// Mitsubishi GX Works2 project: project   PLC: FX3U/FX3UC
// Okoma

TYPE spindleProfile : STRUCT
  valveUp : BOOL;  (* DO_ Valve to move spindle UP *)
  valveDown : BOOL;  (* DO_ Valve to move spindle DOWN *)
  valveInMan : BOOL;  (* Command from HMI to move spindle IN/OUT work *)
  motorOnMan : BOOL;  (* Command from HMI to switch ON motor *)
  recipeOn : BOOL;  (* Spindle must be ON by Recipe from HMI *)
  recipeUp : BOOL;  (* Spindle must be UP by Recipe from HMI *)
  valveUpMan : BOOL;  (* Command from HMI to move spindle UP *)
  valveDownMan : BOOL;  (* Command from HMI to move spindle DOWN *)
  valveIn : BOOL;  (* DO_ Valve to move spindle IN work *)
  motorOn : BOOL;  (* DO_ Contactor to switch ON motor *)
  sensorUp : BOOL;  (* DI_ Sensor spindle in Top position *)
  sensorDown : BOOL;  (* DI_ Sensor spindle in Bottom position *)
  sensorOut : BOOL;  (* DI_ Sensor spindle position OUT of work *)
END_STRUCT END_TYPE

// global labels: Global_Vars
VAR_GLOBAL
  hmiPar10 AT D200.0 : BOOL;  (* Return after Quick Cut Cycle (0-Off, 1-On) *)
  recipeRollerPresser AT D250.4 : BOOL;
  recipeMotor0 AT D250.5 : BOOL;
  recipeMotor4 AT D250.9 : BOOL;
  recipeMotor5 AT D250.A : BOOL;
  recipeBlower AT D250.B : BOOL;
  recipeBetween2and3 AT D250.F : BOOL;
  recipeSpindle0bit0 AT D251.0 : BOOL;
  recipeSpindle0bit1 AT D251.1 : BOOL;
  safetyCircuiteOk AT M0 : BOOL;
  automaticMode AT M5 : BOOL;
  manualMode AT M6 : BOOL;
  alarmState AT M7 : BOOL;
  attentionState AT M8 : BOOL;
  spindle0NotMiddle AT M10 : BOOL;
  carriageBlockNotChange AT M12 : BOOL;
  spindle0NotChange AT M11 : BOOL;
  motorsProfile AT M40 : BOOL;  (* Motor 1, 2,3 or 5 (saw end) is ON *)
  rollersTransporterAuto AT M30 : BOOL;
  carriageMoving AT M20 : BOOL;
  machineBusy AT M9 : BOOL;  (* Excecutung automatic cycle *)
  manCarriageMoveToSensor4 AT M24 : BOOL;
  manCarriageMoveToSensor1 AT M25 : BOOL;
  rollersTransporterContinousMan AT M31 : BOOL;
  thermicOk AT X000 : BOOL;
  controlVoltageOk AT X001 : BOOL;
  airPressureOk AT X002 : BOOL;
  bypassKey AT X003 : BOOL;
  buttonQuickCut AT X010 : BOOL;
  buttonPositioningSpindles AT X017 : BOOL;  (* button S3 *)
  buttonStart2 AT X020 : BOOL;
  carriageSensor1 AT X021 : BOOL;
  carriageSensor2 AT X022 : BOOL;
  carriageSensor3 AT X023 : BOOL;
  carriageSensor4 AT X024 : BOOL;
  pieceInStart AT X025 : BOOL;
  pieceInEnd AT X026 : BOOL;
  buttonStartMotors AT X027 : BOOL;  (* button S60 *)
  buttonAuto AT X030 : BOOL;  (* button S55 *)
  buttonPress AT X031 : BOOL;  (* button S54 *)
  buttonStart AT X032 : BOOL;  (* button S53 *)
  buttonEnable AT X033 : BOOL;  (* button S61 *)
  buttonTransporterForward AT X034 : BOOL;  (* button S62 *)
  buttonTransporterBackward AT X035 : BOOL;  (* button S63 *)
  buttonCarriageForward AT X036 : BOOL;  (* button S36 *)
  buttonCarriageBackward AT X037 : BOOL;  (* button S37 *)
  carriageMoveEnable AT Y001 : BOOL;
  carriageMotorForward AT Y002 : BOOL;
  carriageMotorBackward AT Y003 : BOOL;
  carriageMotorBrake AT Y004 : BOOL;  (* Brake resistor *)
  carriageSpeedWork AT Y005 : BOOL;
  carriageSpeedSlow AT Y006 : BOOL;
  carriageSpeedFast AT Y007 : BOOL;
  spindleMotor0 AT Y010 : BOOL;  (* Motor 0 *)
  sawCarriageMotor AT Y014 : BOOL;  (* Motor 4 *)
  sawEndMotor AT Y015 : BOOL;  (* Motor 5 *)
  transporterMotorBackward AT Y016 : BOOL;
  transporterMotorForward AT Y017 : BOOL;
  pressCarriageValveDown AT Y020 : BOOL;
  spindle0Valve1Up AT Y024 : BOOL;
  spindle0Valve1Down AT Y025 : BOOL;
  spindle0Valve2Up AT Y026 : BOOL;
  spindle0Valve2Down AT Y027 : BOOL;
  pressCarriageValveUp AT Y030 : BOOL;
  pressRollerReleaseValve AT Y037 : BOOL;
  between2and3Valve AT Y040 : BOOL;
  blower AT Y041 : BOOL;
  sawEndValveDown AT Y042 : BOOL;
  lightAlarm AT Y044 : BOOL;
  lightCycleRun AT Y045 : BOOL;  (* Automatic Cycle running White indicator *)
  lightAttention AT Y046 : BOOL;
  PLC_Run AT M8000 : BOOL;
  PLC_getErrors AT M8004 : BOOL;
  carriageNeedForward AT M27 : BOOL;
  carriageNeedBackward AT M28 : BOOL;
  Alarm52 AT D5.2 : BOOL;  (* Alarm: Start Automtic cycle with all motors off *)
  Alarm53 AT D5.3 : BOOL;  (* Alarm: Piece not fixed on carriage by press *)
  Alarm54 AT D5.4 : BOOL;  (* Alarm: Change state motors while some cycle is running *)
  Alarm55 AT D5.5 : BOOL;  (* Alarm: Start motors not in Automatic mode *)
  Alarm46 AT D4.6 : BOOL;  (* Alarm: Too long time Carriage moving backward *)
  Alarm01 AT D0.1 : BOOL;  (* Alarm: Thermic breakers KO *)
  Alarm02 AT D0.2 : BOOL;  (* Alarm: Low air pressure *)
  Alarm03 AT D0.3 : BOOL;  (* Alarm: Control voltage KO *)
  Alarm04 AT D0.4 : BOOL;  (* Alarm: Stop button pressed *)
  Alarm09 AT D0.9 : BOOL;  (* Alarm: Bypass key switched on *)
  Alarm11 AT D1.1 : BOOL;  (* Alarm: Spindle 1 Top and buttom sensors ON *)
  Alarm12 AT D1.2 : BOOL;  (* Alarm: Spindle 1 not in horisontal position *)
  Alarm13 AT D1.3 : BOOL;  (* Alarm: Spindle 1 not in vertical position *)
  Alarm21 AT D2.1 : BOOL;  (* Alarm: Spindle 2 Top and Buttom sensors ON *)
  Alarm22 AT D2.2 : BOOL;  (* Alarm: Spindle 2 not in horisontal position *)
  Alarm23 AT D2.3 : BOOL;  (* Alarm: Spindle 2 not in vertical position *)
  Alarm31 AT D3.1 : BOOL;  (* Alarm: Spindle 3 Top and buttom sensors ON *)
  Alarm32 AT D3.2 : BOOL;  (* Alarm: Spindle 3 Not in horisontal position *)
  Alarm33 AT D3.3 : BOOL;  (* Alarm: Spindle 3 Not in vertical position *)
  Alarm40 AT D4.0 : BOOL;  (* Alarm: More than one carriage sensor ON in one time *)
  Alarm45 AT D4.5 : BOOL;  (* Alarm: Too long time Carriage moving forward *)
  Alarm56 AT D5.6 : BOOL;  (* Alarm: Positioning spindles not in Automatic mode *)
  Alarm47 AT D4.7 : BOOL;  (* Alarm: Move carriage with Spindle 0 in middle *)
  Alarm58 AT D5.8 : BOOL;  (* Alarm: Positioning spindles 0 with block change and piece pressed *)
  Alarm59 AT D5.9 : BOOL;  (* Alarm: Positioning spindles 0 in carriage unknown position *)
  Alarm50 AT D5.0 : BOOL;  (* Alarm: Positionig cycle by pneumatic not finished *)
  Alarm51 AT D5.1 : BOOL;  (* Alarm: Start motors cycle not finished *)
  motorsDovetail AT M41 : BOOL;  (* Motor 0 or 4 (saw carriage) is ON *)
  Alarm57 AT D5.7 : BOOL;  (* Alarm: Positioning spindles while some cycle is running *)
  Alarm5A AT D5.A : BOOL;  (* Alarm: Start cycle not in Automatic mode *)
  Alarm5C AT D5.C : BOOL;  (* Alarm: Start Automatic cycle while another cycle is running *)
  PLC_InitialPulse AT M8002 : BOOL;
  Alarm48 AT D4.8 : BOOL;  (* Alarm: Move carriage backward with Sensor 1 On *)
  Alarm49 AT D4.9 : BOOL;  (* Alarm: Move carriage forward with Sensor 4 On *)
  plcRunTime AT D10 : TIME;  (* PLC running time in ms (step 10 ms) *)
  hmiPar11 AT D200.1 : BOOL;  (* Cut (0-slow, 1-quick) *)
  workTime AT D230 : DINT;  (* Time machine run (in seconds) *)
  hmiPar1 AT D201 : TIME;  (* Delay to slowdown carriage (0..5sec) *)
  hmiPar2 AT D203 : TIME;
  hmiPar3 AT D205 : TIME;  (* Delay carriage presser release (0..1sec) *)
  hmiPar4 AT D207 : TIME;  (* Delay blower OFF (0..60sec) *)
  hmiPar5 AT D209 : TIME;  (* Delay Off Roller Transporter (0..60sec) *)
  hmiPar6 AT D211 : TIME;  (* Safety max time carriage moving (0..60sec) *)
  stepAuto AT D21 : INT;  (* Step of Automatic cycle *)
  carriageAutoForward AT M21 : BOOL;
  carriageAutoBackward AT M22 : BOOL;
  Alarm41 AT D4.1 : BOOL;  (* Alarm: Carriage sensor 1 not working *)
  Alarm42 AT D4.2 : BOOL;  (* Alarm: Carriage sensor 2 not working *)
  Alarm43 AT D4.3 : BOOL;  (* Alarm: Carriage sensor 3 not working *)
  Alarm44 AT D4.4 : BOOL;  (* Alarm: Carriage sensor 4 not working *)
  carriageSpeed AT D20 : INT;  (* Carriage speed (1-Slow, 3-Fast, 5-Work/Mill) *)
  pulseEvery1sec AT M8013 : BOOL;
  pulseEvery10msec AT M8011 : BOOL;
  stepStartMotors AT D22 : INT;  (* Step of motors start cycle *)
  stepPneumaticPositioning AT D23 : INT;  (* Step of pneumatic positioning cycle *)
  sensorPositionPrev AT D24 : INT;  (* Previous detected carriage position *)
  sensorPositionCurrent AT D25 : INT;  (* Current carriage position *)
  spindle0Valve1UpMemory AT D232.1 : BOOL;  (* Save state spindle 0 valve 0 *)
  spindle0Valve2UpMemory AT D232.2 : BOOL;  (* Save state spindle 0 valve 1 *)
  PLC_LithiumBatteryKO AT M8005 : BOOL;
  PLC_PowerKO AT M8007 : BOOL;
  presserCarriageValveUpMemory AT D232.0 : BOOL;  (* Save state carriage presser *)
  Alarm5B AT D5.B : BOOL;  (* Alarm: Button carriage move not in Manual mode *)
  Alarm5D AT D5.D : BOOL;  (* Alarm: Button rollers transporter move not in Manual mode *)
  Alarm5E AT D5.E : BOOL;  (* Alarm: Button Start2 with motors 1-2-3-5 OFF *)
  speedCut AT D26 : INT;  (* Speed carriage cut *)
  speedMill AT D27 : INT;  (* Speed carriage mill *)
END_VAR
VAR_GLOBAL CONSTANT
  distanceS1S2 : INT := 532;  (* Distance between carriage MEF(Sensor1) and MEF(Sensor2), mm *)
  distanceS2S3 : INT := 454;  (* Distance between carriage MEF(Sensor2) and MEP(Sensor3), mm *)
END_VAR
VAR_GLOBAL
  plcRunTime2 AT D12 : DINT;  (* PLC running time in ms (step 10 ms) *)
  pulseEvery100msec AT M8012 : BOOL;
  pressRollerMan AT M116 : BOOL;  (* HMI Press Roller in Manual mode *)
  blowerMan AT M117 : BOOL;  (* HMI Blower in Manual mode *)
  spindleMotor0Man AT M130 : BOOL;  (* HMI Spindle 0 Motor in Manual mode *)
  spindleMotor4Man AT M134 : BOOL;  (* HMI Spindle 4 Motor in Manual mode *)
  spindleMotor5Man AT M135 : BOOL;  (* HMI Spindle 5 Motor in Manual mode *)
  spindle0Valve1UpMan AT M110 : BOOL;  (* HMI Spindle 0 Valve 1 Up in Manual mode *)
  spindle0Valve1DownMan AT M111 : BOOL;  (* HMI Spindle 0 Valve 1 Down in Manual mode *)
  spindle0Valve2UpMan AT M112 : BOOL;  (* HMI Spindle 0 Valve 2 Up in Manual mode *)
  spindle0Valve2DownMan AT M113 : BOOL;  (* HMI Spindle 0 Valve 2 Down in Manual mode *)
  between2and3ValveMan AT M118 : BOOL;  (* HMI Block between spindle 2 and 3 Valve in Manual mode *)
  sawEndValveMan AT M115 : BOOL;  (* HMI Saw End after spindle 3 Valve in Manual mode *)
  spindle1 : spindleProfile;
  spindle2 : spindleProfile;
  spindle3 : spindleProfile;
END_VAR

// task MAIN (event TRUE, interval 0, priority 30): Automatic_Cycles, Carriage, Spindles_Motors, Roller_Transporter, Pneumatic_Positioning, Main
// task Alarms (event TRUE, interval 0, priority 31): Alarms

PROGRAM VFD_Modbus
VAR
  errorsCode : INT;
  errorBit : BOOL;
  errorsCount : INT;
  atvReset_inProgress : BOOL;
  atvWriteSpeed_inProgress : BOOL;
  atvForward_inProgress : BOOL;
  atvBackward_inProgress : BOOL;
  atvReset_inQueue : BOOL;
  atvWriteSpeed_inQueue : BOOL;
  atvForward_inQueue : BOOL;
  atvBackward_inQueue : BOOL;
  channelBussy : BOOL;
  TOFdelay : TOF_10;
  atvShutdown_inQueue : BOOL;
  atvShutdown_inProgress : BOOL;
  atvReadData_inProgress : BOOL;
  atvReadData_inQueue : BOOL;
  counter : INT;
  RS2running : BOOL;
  timeRS2 : INT;
END_VAR
IF M8002 THEN
    D8400 := H1C87; (* Параметры связи для команды RS2 через Ch1 *) (* 0001 1100 1000 0111 -> 9600 8E1 *)
    D8409 := K10; (* Задержка включения флагов M8409 и M8403 при НЕ получении ответа: 10x10 = 100ms *)
    M8161 := FALSE; (* data bit length TRUE-8bit, FALSE-16bit *)
    ZRST(TRUE , D300 , D303); (* Очистка памяти отправляемых данных *)
    ZRST(TRUE , D310 , D313); (* Очистка памяти принимаемых данных*)
    errorsCount := 0; (* Очистка счётчика ошибок *)
END_IF;

errorBit := M8063; (* M8063 включается при ошибке связи *)
errorsCode := D8063; (* D8063 хранит код ошибки связи *)

(* Заносим команды в очередь - inQueue *)
SET ( MEF(buttonEnable), atvReset_inQueue); (* Сброс аварийного состояния частотника *)
SET ( MEP(carriageMoveEnable) OR MEF(carriageMoveEnable), atvShutdown_inQueue); (* Переход в режим READY_TO_SWITCH_ON перед запуском или при остановке *)
SET ( MEP( carriageSpeedSlow) OR MEP (carriageSpeedWork) OR MEP(carriageSpeedFast), atvWriteSpeed_inQueue); (* Смена скорости *)
SET ( MEP(carriageMotorForward), atvForward_inQueue); (* Движение вперёд *)
SET ( MEP(carriageMotorBackward), atvBackward_inQueue); (* Движение назад *)
SET ( MEP(M8013), atvReadData_inQueue); (* Запрашивать состояние частотника каждую секунду *)

(* Измерение времени работы команды RS2 *)
SET(MEP(M8402), RS2running);
RST(MEP(M8403), RS2running);
IF RS2running THEN counter := counter + 1; END_IF; (* Счётчик циклов работы команды RS2 *)
IF MEP(M8403) THEN
	timeRS2 := counter * D8010; (* Время x0.1мс работы команды RS2 *)
	counter := 0;
END_IF;


TOFdelay ( IN:= M8402 , PT:=T#50ms, Q:=channelBussy); (* Минимальное время между отправкой команд *)
(* При задержке меньше 30 мс возникают ошибки *)

RS2 ( atvReadData_inProgress, D300, K8, K7, K1, D310); (* Команда для чтения данных из частотника (пакет 7 байт) *)
RS2 ( NOT atvReadData_inProgress, D300, K8, K8, K1, D310); (* Команда записи данных в частотник (пакет 8 байт) *)

IF MEP(M8403) THEN
	M8403 := FALSE; (* Перед отправкой очередного пакета необходимо сбросить M8403 *)
	IF (D300=H0601 AND D303=D313) OR (D300=H0301 AND D300=D310) THEN (* Проверка отправленного и полученного CRC *)
		IF atvReset_inProgress THEN
			atvReset_inQueue := FALSE;
			M8063 := FALSE; (* Сброс бита ошибки передачи данных *)
			D8063 := 0; (* Сброс кода ошибки передачи данных *)
		END_IF;
		RST(atvShutdown_inProgress, atvShutdown_inQueue);
	 	RST(atvWriteSpeed_inProgress, atvWriteSpeed_inQueue);
	 	RST(atvForward_inProgress, atvForward_inQueue);
	 	RST(atvBackward_inProgress, atvBackward_inQueue);
	 	RST(atvReadData_inProgress, atvReadData_inQueue);
	ELSE
	 	errorsCount := errorsCount + 1;
	END_IF;
	atvReset_inProgress := FALSE;
	atvShutdown_inProgress := FALSE;
	atvWriteSpeed_inProgress := FALSE;
	atvForward_inProgress := FALSE;
	atvBackward_inProgress := FALSE;
	atvReadData_inProgress := FALSE;
	(*ZRST(TRUE , D310 , D313);*)
END_IF;

(* FAULT RESET - Сброс ошибок частотника *)
IF atvReset_inQueue AND NOT M8402 AND NOT channelBussy AND NOT M8403 THEN
	atvShutdown_inQueue := FALSE;
	atvForward_inQueue := FALSE;
	atvBackward_inQueue := FALSE;
	atvReadData_inQueue := FALSE;
    D300 := H0601; (* 01 Slave adress, 06 Code write word *)
    D301 := H3521; (* K8501 Control word address *)
    D302 := H8000; (* H80 FAULT RESET *)
    CRC( TRUE , D300 , K6 , D303 );
	M8402 := TRUE; (* Start sending package to ATV*)
	atvReset_inProgress := TRUE; (* RESET command was send *)
END_IF;

(* SHUTDOWN - Необходимо выполнить перед запуском и при остановке *)
IF atvShutdown_inQueue AND NOT M8402 AND NOT channelBussy AND NOT M8403 THEN
	atvForward_inQueue := FALSE;
	atvBackward_inQueue := FALSE;
    D300 := H0601; (* 01 Slave adress, 06 Code write word *)
    D301 := H3521; (* K8501 Control word address *)
    D302 := H0600; (* H6 SHUT DOWN *)
    CRC( TRUE , D300 , K6 , D303 );
	M8402 := TRUE;
	atvShutdown_inProgress := TRUE;
END_IF;

(* WRITE SPEED - Задание скорости *)
IF atvWriteSpeed_inQueue AND NOT M8402 AND NOT channelBussy AND NOT M8403 THEN
    D300 := H0601; (* 01 Slave adress, 06 Code write word *)
    D301 := H3621; (* K8502 Control word address *)
    IF carriageSpeedSlow THEN D302 := K120; (* 12.0 Hz  *)
    	ELSIF carriageSpeedWork THEN D302 := K200;
    	ELSIF carriageSpeedFast THEN D302 := K600;
    	ELSE D302 := 0;
    END_IF;
	SWAP(TRUE, D302);
    CRC( TRUE , D300 , K6 , D303 );
	M8402 := TRUE; (* Start sending package to ATV *)
	atvWriteSpeed_inProgress := TRUE; (* Команда смены скорости отправлена *)
END_IF;

(* ENABLE OPERATION - FORWARD - Вращение вперёд *)
IF atvForward_inQueue AND NOT M8402 AND NOT channelBussy AND NOT M8403 THEN
    D300 := H0601; (* 01 Slave adress, 06 Code write word *)
    D301 := H3521; (* K8501 Control word address *)
    D302 := H0F00; (* HF ENABLE OPERATION *)
    CRC( TRUE , D300 , K6 , D303 );
	M8402 := TRUE; (* Start sending package to ATV*)
	atvForward_inProgress := TRUE; (* Команда FORWARD отправлена *)
END_IF;

(* ENABLE OPERATION - BACKWARD - Вращение назад *)
IF atvBackward_inQueue AND NOT M8402 AND NOT channelBussy AND NOT M8403 THEN
    D300 := H0601; (* 01 Slave adress, 06 Code write word *)
    D301 := H3521; (* K8501 Control word address *)
    D302 := H0F08; (* K2063 RUN BACKWARD *)
    CRC( TRUE , D300 , K6 , D303 );
	M8402 := TRUE; (* Start sending package to ATV*)
	atvBackward_inProgress := TRUE; (* Команда BACKWARD отправлена *)
END_IF;

(* READ DATA - Чтение данных из памяти частотника *)
IF atvReadData_inQueue AND NOT M8402 AND NOT channelBussy AND NOT M8403 THEN
    D300 := H0301; (* 1byte - 01 Slave adress, 2byte - 03 Code read words *)
    D301 := H3521; (* Control word address: 2bytes PLC Lo-Hi H3521 -> VFD Modbus Hi-Lo H2135=K8501 *)
    D302 := H0100; (* Number of words: 2bytes PLC Lo-Hi H0100 -> Modbus VFD Hi-Lo H0001*)
    CRC( TRUE , D300 , K6 , D303 );
	M8402 := TRUE;
	atvReadData_inProgress := TRUE;
END_IF;
END_PROGRAM

FUNCTION crc_my
VAR_INPUT
  Word0 : WORD;
  Word1 : WORD;
  Word2 : WORD;
END_VAR
VAR
  counterWords : INT;
  counterByte : INT;
  counterBit : INT;
  lsb : BOOL;
  dataArray : ARRAY [0..2] OF WORD;
  dataWord : WORD;
  dataByte : ARRAY [0..1] OF WORD;
  crcCalc : WORD;
END_VAR
(* Заносим слова в массив для обработки в цикле*)
dataArray[0] := Word0;
dataArray[1] := Word1;
dataArray[2] := Word2;

crcCalc := HFFFF; (* Начальный полином *)

FOR counterWords:=0 TO 2 DO (* Перебираем слова в массиве dataArray*)
	dataWord := dataArray[counterWords];
	WTOB(TRUE , dataWord , 2 , dataByte[0]); (* Делим слово dataWord на 2 байта и заносим в массив dataByte*)

	FOR counterByte:=0 TO 1 DO (*Перебираем байты слова *)
		crcCalc := crcCalc XOR dataByte[counterByte];
		FOR counterBit:=1 TO 8 DO (*Перебираем и сдвигаем биты однго байта*)
			BON(TRUE , crcCalc, 0, lsb); (* Получаем первый бит *)
			IF  lsb THEN (* Если первый бит = 1 *)
				crcCalc := SHR(crcCalc,1);
				crcCalc := crcCalc XOR HA001;
			ELSE
				crcCalc := SHR(crcCalc,1);
			END_IF;
		END_FOR;
	END_FOR;
	
END_FOR;
crc_my := crcCalc; (* Возврат результата *)
END_FUNCTION

PROGRAM Main
(* Запись времени работы ПЛК с дискретностью 10 мс *)
IF MEP(pulseEvery10msec) THEN
	plcRunTime := plcRunTime + T#10ms;
END_IF;

(* Запись времени работы ПЛК с дискретностью равной времени цикла ПЛК (D8010) *)
(*plcRunTime2 := plcRunTime2 + WORD_TO_DINT(D8010);*)

(* Запись времени работы станка с дискретностью 1 с *)
IF MEP(pulseEvery1sec) AND
	(machineBusy OR motorsDovetail OR motorsProfile OR carriageMoveEnable OR transporterMotorForward OR transporterMotorBackward) THEN
	workTime := workTime + 1;
END_IF;

(* Replace parameters values If battery fail or memory cleared*)
IF hmiPar5=T#0s THEN
	hmiPar5 := T#10s;
END_IF;

IF hmiPar6=T#0s THEN
	hmiPar6 := T#60s;
END_IF;

(* Цепочка безопасности *)
safetyCircuiteOk := PLC_Run AND NOT PLC_getErrors AND ((thermicOk AND airPressureOk AND controlVoltageOk)  OR bypassKey);

(* Режим работы Ручной/Автоматический *)
automaticMode := buttonAuto;
manualMode := NOT buttonAuto;


(* Сохранение состояний пневматических клапанов при отключении питания ПЛК *)
IF PLC_PowerKO THEN
	presserCarriageValveUpMemory := pressCarriageValveUp;
	spindle0Valve1UpMemory := spindle0Valve1Up;
	spindle0Valve2UpMemory := spindle0Valve2Up;
END_IF;

(* Восстановление состояний пневматичесих клапанов после включения ПЛК *)
IF PLC_InitialPulse THEN
	pressCarriageValveUp := presserCarriageValveUpMemory;
	pressCarriageValveDown := NOT pressCarriageValveUp;

	spindle0Valve1Up := spindle0Valve1UpMemory;
	spindle0Valve1Down := NOT spindle0Valve1Up;
	
	spindle0Valve2Up := spindle0Valve2UpMemory;
	spindle0Valve2Down := NOT spindle0Valve2Up;
END_IF;
END_PROGRAM

FUNCTION_BLOCK FB_DOUBLE_CLICK
VAR_INPUT
  PERIOD : TIME;
END_VAR
VAR_OUTPUT
  Q : BOOL;
END_VAR
VAR
  timeClickBefore : TIME;
END_VAR
VAR_INPUT
  IN : BOOL;
END_VAR
IF MEP(IN) THEN
	Q := ((plcRunTime-timeClickBefore) > T#10ms) AND ((plcRunTime-timeClickBefore) < PERIOD);
	timeClickBefore := plcRunTime;
END_IF;

IF NOT Q	THEN
	RETURN;
ELSIF (plcRunTime - timeClickBefore) > PERIOD THEN
	Q := FALSE;
END_IF;
END_FUNCTION_BLOCK

PROGRAM Spindles_Motors
VAR
  TONDelay : TON;  (* Alarm: Change state motors while some cycle is running *)
  varOut : TIME;
  stepFirstRun : BOOL;
END_VAR
IF NOT buttonEnable OR NOT safetyCircuiteOk OR MEF(manualMode) THEN
	stepStartMotors := 0;
	spindleMotor0 := FALSE;
	spindle1.motorOn := FALSE;
	spindle2.motorOn := FALSE;
	spindle3.motorOn := FALSE;
	sawCarriageMotor := FALSE;
	sawEndMotor := FALSE;
END_IF;

IF MEP(buttonStartMotors) AND stepStartMotors=0 THEN
	IF automaticMode AND NOT machineBusy THEN
		stepStartMotors := 10;
	ELSE
		SET(machineBusy, Alarm54);
		SET(NOT automaticMode, Alarm55);
	END_IF;
END_IF;

RST(NOT machineBusy, Alarm54);
RST(automaticMode, Alarm55);

(* Цикл запуска моторов *)
CASE stepStartMotors OF
	0:
		stepFirstRun := TRUE;
		TONDelay(IN := FALSE);
		Alarm51 := FALSE;

	10: (* Активация цикла запуска мотора 0 - Шпиндель 0 *)
		TONDelay.IN := FALSE;
		IF (stepFirstRun AND (spindleMotor0 OR NOT recipeMotor0)) OR TONDelay.Q THEN
			stepStartMotors := 11;
			stepFirstRun := TRUE;
		ELSE
			stepFirstRun := FALSE;
			TONDelay.IN := TRUE;
		END_IF;
		spindleMotor0 := recipeMotor0;
		TONDelay(PT:=T#8s, ET:= varOut);

	11: (* Активация цикла запуска мотора 1 - Шпиндель 1 *)
		TONDelay.IN := FALSE;
		IF (stepFirstRun AND (spindle1.motorOn OR NOT spindle1.recipeOn)) OR TONDelay.Q THEN
			stepStartMotors := 12;
			stepFirstRun := TRUE;
		ELSE
			stepFirstRun := FALSE;
			TONDelay.IN := TRUE;
		END_IF;
		spindle1.motorOn := spindle1.recipeOn;
		TONDelay(PT:=T#4s);
		
	12: (* Активация цикла запуска мотора 2 - Шпиндель 2 *)
		TONDelay.IN := FALSE;
		IF (stepFirstRun AND (spindle2.motorOn OR NOT spindle2.recipeOn)) OR TONDelay.Q THEN
			stepStartMotors := 13;
			stepFirstRun := TRUE;
		ELSE
			stepFirstRun := FALSE;
			TONDelay.IN := TRUE;
		END_IF;
		spindle2.motorOn := spindle2.recipeOn;
		TONDelay(PT:=T#4s);

	13: (* Активация цикла запуска мотора 3 - Шпиндель 3 *)
		TONDelay.IN := FALSE;
		IF (stepFirstRun AND (spindle3.motorOn OR NOT spindle3.recipeOn)) OR TONDelay.Q THEN
			stepStartMotors := 14;
			stepFirstRun := TRUE;
		ELSE
			stepFirstRun := FALSE;
			TONDelay.IN := TRUE;
		END_IF;
		spindle3.motorOn := spindle3.recipeOn;
		TONDelay(PT:=T#4s);

	14: (* Активация цикла запуска мотора 4 - Торцовка каретки *)
		TONDelay.IN := FALSE;
		IF (stepFirstRun AND (sawCarriageMotor OR NOT recipeMotor4 OR sawEndMotor OR NOT recipeMotor5)) OR TONDelay.Q THEN
			stepStartMotors := 15;
		ELSE
			stepFirstRun := FALSE;
			TONDelay.IN := TRUE;
		END_IF;
		sawCarriageMotor := recipeMotor4;
		TONDelay(PT:=T#2s);

	15: (* Активация цикла запуска мотора 5 - Пила после 3-го шпинделя *)
		sawEndMotor := recipeMotor5;
		stepStartMotors := 0;
END_CASE;


(* Управление моторами шпинделей в ручном режиме *)
IF manualMode THEN
	IF MEP(spindleMotor0Man) THEN spindleMotor0 := INV(spindleMotor0); END_IF;
	IF MEP(spindle1.motorOnMan) THEN spindle1.motorOn := INV(spindle1.motorOn); END_IF;
	IF MEP(spindle2.motorOnMan) THEN spindle2.motorOn := INV(spindle2.motorOn); END_IF;
	IF MEP(spindle3.motorOnMan) THEN spindle3.motorOn := INV(spindle3.motorOn); END_IF;
	IF MEP(spindleMotor4Man) THEN sawCarriageMotor := INV(sawCarriageMotor); END_IF;
	IF MEP(spindleMotor5Man) THEN sawEndMotor := INV(sawEndMotor); END_IF;
END_IF;
	
motorsProfile := spindle1.motorOn OR spindle2.motorOn OR spindle3.motorOn OR sawEndMotor;
motorsDovetail :=  spindleMotor0 OR sawCarriageMotor;
END_PROGRAM

PROGRAM Pneumatic_Positioning
IF NOT buttonEnable OR NOT safetyCircuiteOk  OR NOT automaticMode THEN
	stepPneumaticPositioning := 0;
	(*between2and3Valve := FALSE;
	sawEndValveDown := FALSE;*)
END_IF;

(* Запуск цикла позиционирования узлов на пневматике *)
IF MEP(buttonPositioningSpindles) THEN
	IF automaticMode AND safetyCircuiteOk AND NOT machineBusy THEN
		stepPneumaticPositioning := 5;
	ELSE
		SET(NOT automaticMode, Alarm56);
		SET(machineBusy, Alarm57);
	END_IF;
END_IF;

RST(spindle0NotMiddle, Alarm47);
RST(automaticMode, Alarm56);
RST(NOT machineBusy, Alarm57);
RST(pressCarriageValveUp, Alarm58);
RST(carriageSensor1 OR carriageSensor2 OR carriageSensor3 OR carriageSensor4, Alarm59);

(* Упор каретки не меняет положения при заданном рецепте *)
carriageBlockNotChange := spindle0Valve1Up XOR recipeSpindle0bit1;

(* Шпиндель 0 не меняет вертикальное положение *)
spindle0NotChange := (spindle0Valve1Down=recipeSpindle0bit1) AND (spindle0Valve2Down=recipeSpindle0bit0);

(* Шпиндель 0 НЕ в среднем положении *)
spindle0NotMiddle := (spindle0Valve1Up AND spindle0Valve2Up) OR (spindle0Valve1Down AND spindle0Valve2Down);


(* Цикл позиционирования узлов *)
CASE stepPneumaticPositioning OF
	0:
		Alarm50 := FALSE;

	5: (* Позиционирование шпинделя 0 *)
		IF NOT spindle0NotChange THEN
			IF (carriageSensor1 OR carriageSensor2 OR carriageSensor3 OR carriageSensor4) AND (carriageBlockNotChange OR pressCarriageValveUp) THEN
				IF NOT recipeSpindle0bit0 AND NOT recipeSpindle0bit1 THEN (* Шпиндель 0 - Положение верхнее, Упор 1 *)
					spindle0Valve1Up := TRUE; spindle0Valve1Down := NOT spindle0Valve1Up;
					spindle0Valve2Up := TRUE; spindle0Valve2Down := NOT spindle0Valve2Up;
				ELSIF recipeSpindle0bit0 AND NOT recipeSpindle0bit1 THEN (* Шпиндель 0 - Положение среднее, Упор 1 *)
					spindle0Valve1Up := TRUE; spindle0Valve1Down := NOT spindle0Valve1Up;
					spindle0Valve2Up := FALSE; spindle0Valve2Down := NOT spindle0Valve2Up;
				ELSIF NOT recipeSpindle0bit0 AND recipeSpindle0bit1 THEN (* Шпиндель 0 - Положение среднее, Упор 2 *)
					spindle0Valve1Up := FALSE; spindle0Valve1Down := NOT spindle0Valve1Up;
					spindle0Valve2Up := TRUE; spindle0Valve2Down := NOT spindle0Valve2Up;
				ELSIF recipeSpindle0bit0 AND recipeSpindle0bit1 THEN (* Шпиндель 0 - Положение нижнее, Упор 2 *)
					spindle0Valve1Up := FALSE; spindle0Valve1Down := NOT spindle0Valve1Up;
					spindle0Valve2Up := FALSE; spindle0Valve2Down := NOT spindle0Valve2Up;
				END_IF;
			ELSE
				SET(NOT carriageBlockNotChange AND NOT pressCarriageValveUp, Alarm58);
				SET(NOT carriageSensor1 AND NOT carriageSensor2 AND NOT carriageSensor3 AND NOT carriageSensor4, Alarm59);
			END_IF;
		END_IF;
		stepPneumaticPositioning := 7;

	7:
		between2and3Valve := recipeBetween2and3; (* Упор между 2-м и 3-м шпинделями *)
		sawEndValveDown := recipeMotor5; (* Пила после 3-го шпинделя - Мотор 5 *)
		stepPneumaticPositioning := 10;

	10: (* Возвращение шпинделей 1-2-3 в исходное горизонтальное положение. Только для шпинделей, которые выключаются или меняют вертикальное положение *)
		RST(((spindle1.valveIn AND NOT spindle1.recipeOn) OR (spindle1.valveUp XOR spindle1.recipeUp)) AND (spindle1.sensorUp XOR spindle1.sensorDown), spindle1.valveIn);
		RST(((spindle2.valveIn AND NOT spindle2.recipeOn) OR (spindle2.valveUp XOR spindle2.recipeUp)) AND (spindle2.sensorUp XOR spindle2.sensorDown), spindle2.valveIn);
		RST(((spindle3.valveIn AND NOT spindle3.recipeOn) OR (spindle3.valveUp XOR spindle3.recipeUp)) AND (spindle3.sensorUp XOR spindle3.sensorDown), spindle3.valveIn);

		IF (spindle1.valveIn XOR spindle1.sensorOut) AND (spindle2.valveIn XOR spindle2.sensorOut) AND (spindle3.valveIn XOR spindle3.sensorOut) THEN
			stepPneumaticPositioning := 20; END_IF;
	
	20: (* Вертикальное позиционирование шпинделей 1-2-3. Только для шпинделей, которые включены по рецепту и меняют вертикальное положение *)
		IF spindle1.sensorOut AND spindle1.recipeOn THEN
			spindle1.valveUp := spindle1.recipeUp;
			spindle1.valveDown := NOT spindle1.valveUp; END_IF;
		IF spindle2.sensorOut AND spindle2.recipeOn THEN
			spindle2.valveUp := spindle2.recipeUp;
			spindle2.valveDown := NOT spindle2.valveUp; END_IF;
		IF spindle3.sensorOut AND spindle3.recipeOn THEN
			spindle3.valveUp := spindle3.recipeUp;
			spindle3.valveDown := NOT spindle3.valveUp; END_IF;
			
		IF ((spindle1.valveUp AND spindle1.sensorUp) OR (spindle1.valveDown AND spindle1.sensorDown) OR (NOT spindle1.valveUp AND NOT spindle1.valveDown)) AND
			 ((spindle2.valveUp AND spindle2.sensorUp) OR (spindle2.valveDown AND spindle2.sensorDown) OR (NOT spindle2.valveUp AND NOT spindle2.valveDown)) AND
			 ((spindle3.valveUp AND spindle3.sensorUp) OR (spindle3.valveDown AND spindle3.sensorDown) OR (NOT spindle3.valveUp AND NOT spindle3.valveDown)) THEN
			 stepPneumaticPositioning := 30; END_IF;

	30: (* Горизонтальное перемещение шпинделей	вперёд. Только для шпинделей, которые включены по рецепту *)
		SET(spindle1.recipeOn AND (spindle1.sensorUp XOR spindle1.sensorDown), spindle1.valveIn);
		SET(spindle2.recipeOn AND (spindle2.sensorUp XOR spindle2.sensorDown), spindle2.valveIn);
		SET(spindle3.recipeOn AND (spindle3.sensorUp XOR spindle3.sensorDown), spindle3.valveIn);

		IF (spindle1.valveIn XOR spindle1.sensorOut) AND (spindle2.valveIn XOR spindle2.sensorOut) AND (spindle3.valveIn XOR spindle3.sensorOut) THEN
			stepPneumaticPositioning := 0; END_IF;
			
END_CASE;

(* РУЧНОЕ УПРАВЛЕНИЕ КЛАПАНАМИ *)
IF manualMode THEN
	(* Ручное управление клапанами шпинделя 0 *)
	IF MEP(spindle0Valve1UpMan) THEN
		spindle0Valve1Up := TRUE;
		spindle0Valve1Down := NOT spindle0Valve1Up; END_IF;
	IF MEP(spindle0Valve1DownMan) THEN
		spindle0Valve1Up := FALSE;
		spindle0Valve1Down := NOT spindle0Valve1Up; END_IF;
	IF MEP(spindle0Valve2UpMan) THEN
		spindle0Valve2Up := TRUE;
		spindle0Valve2Down := NOT spindle0Valve2Up; END_IF;
	IF MEP(spindle0Valve2DownMan) THEN
		spindle0Valve2Up := FALSE;
		spindle0Valve2Down := NOT spindle0Valve2Up; END_IF;

	(* Ручное управление клапанами шпинделя 1 *)
	IF MEP(spindle1.valveUpMan) AND spindle1.sensorOut THEN (* Вверх *)
		spindle1.valveUp := TRUE;
		spindle1.valveDown := NOT spindle1.valveUp; END_IF;
	IF MEP(spindle1.valveDownMan) AND spindle1.sensorOut THEN (* Вниз *)
		spindle1.valveDown := TRUE;
		spindle1.valveUp := NOT spindle1.valveDown; END_IF;
	IF (spindle1.sensorUp XOR spindle1.sensorDown) AND MEP(spindle1.valveInMan) THEN (* Вперёд / Назад *)
		spindle1.valveIn := NOT spindle1.valveIn; END_IF;
		
	(* Ручное управление клапанами шпинделя 2 *)
	IF MEP(spindle2.valveUpMan) AND spindle2.sensorOut THEN
		spindle2.valveUp := TRUE;
		spindle2.valveDown := NOT spindle2.valveUp; END_IF;
	IF MEP(spindle2.valveDownMan) AND spindle2.sensorOut THEN
		spindle2.valveDown := TRUE;
		spindle2.valveUp := NOT spindle2.valveDown; END_IF;
	IF (spindle2.sensorUp XOR spindle2.sensorDown) AND MEP(spindle2.valveInMan) THEN
		spindle2.valveIn := NOT spindle2.valveIn; END_IF;
		
	(* Ручное управление клапанами шпинделя 3 *)
	IF MEP(spindle3.valveUpMan) AND spindle3.sensorOut THEN
		spindle3.valveUp := TRUE;
		spindle3.valveDown := NOT spindle3.valveUp; END_IF;
	IF MEP(spindle3.valveDownMan) AND spindle3.sensorOut THEN
		spindle3.valveDown := TRUE;
		spindle3.valveUp := NOT spindle3.valveDown; END_IF;
	IF (spindle3.sensorUp XOR spindle3.sensorDown) AND MEP(spindle3.valveInMan) THEN
		spindle3.valveIn := NOT spindle3.valveIn; END_IF;

	(* Ручное управление упором между 2-м и 3-м шпинделями *)
	IF MEP(between2and3ValveMan) THEN
		between2and3Valve := NOT between2and3Valve; END_IF;

	(* Ручное управление клапаном пилы после 3-го шпинделя - Мотор 5 *)
	IF MEP(sawEndValveMan) THEN
		sawEndValveDown := NOT sawEndValveDown; END_IF;
END_IF;
END_PROGRAM

PROGRAM Roller_Transporter
VAR
  TOFStopRollerTransporterManF : TOF;  (* Delay OFF Roller Transporter in manual *)
  FB_DOUBLE_CLICK_1 : FB_DOUBLE_CLICK;
  TOFBlower : TOF;
  TOFStopRollerTransporterManB : TOF;  (* Delay OFF Roller Transporter in manual *)
  TOFMotorBackward : TOF;
  TOFMotorForward : TOF;
END_VAR
(* Роликовый транспортёр *)
IF automaticMode THEN
	transporterMotorForward := rollersTransporterAuto;
END_IF;

IF manualMode THEN
	TOFStopRollerTransporterManF(IN:= buttonTransporterForward, PT:= T#1s);
	transporterMotorForward := (TOFStopRollerTransporterManF.Q OR rollersTransporterContinousMan) AND NOT TOFMotorBackward.Q;
	TOFMotorForward(IN:= transporterMotorForward  ,PT:= T#2s);
	
	TOFStopRollerTransporterManB(IN:= buttonTransporterBackward, PT:= T#1s);
	transporterMotorBackward := TOFStopRollerTransporterManB.Q AND NOT TOFMotorForward.Q;
	TOFMotorBackward(IN:= transporterMotorBackward  ,PT:= T#2s);

	FB_DOUBLE_CLICK_1(IN:=MEP(buttonTransporterForward), PERIOD:= T#1s);
	SET(FB_DOUBLE_CLICK_1.Q, rollersTransporterContinousMan);
END_IF;

RST(buttonTransporterForward OR buttonTransporterBackward OR NOT manualMode OR NOT buttonEnable OR NOT safetyCircuiteOk, rollersTransporterContinousMan);

(* Авария - Ручное управление роликовым транспортёром в Автоматическом режиме *)
IF NOT manualMode AND (buttonTransporterBackward OR buttonTransporterForward) THEN
	Alarm5D := TRUE;
END_IF;
RST(manualMode, Alarm5D);

(* ==================================================== *)
(* Прижимные ролики в начале роликового транспортёра *)
IF automaticMode THEN
	pressRollerReleaseValve := TRUE;
	IF (stepAuto=60) AND recipeRollerPresser THEN
		pressRollerReleaseValve := FALSE;
	END_IF;
END_IF;	

IF manualMode AND MEP(pressRollerMan) THEN
	pressRollerReleaseValve := INV( pressRollerReleaseValve );
END_IF;

(* =========================== *)
(* Обдув перед 1-м шпинделем  *)
blower := FALSE;
TOFBlower.IN:= FALSE;
IF automaticMode AND transporterMotorForward AND recipeBlower THEN
	TOFBlower.IN:= pieceInStart;
	blower := TOFBlower.Q;
ELSIF manualMode THEN
	blower := blowerMan;
END_IF;

TOFBlower(PT:= hmiPar4);
END_PROGRAM

PROGRAM Alarms
VAR
  TONspindle1Out : TON;
  TONspindle2Out : TON;
  TONspindle3Out : TON;
  TONspindle1Vertical : TON;
  TONspindle2Vertical : TON;
  TONspindle3Vertical : TON;
END_VAR
(* Сброс аварийных состояний *)
IF NOT buttonEnable THEN
	Alarm11 := FALSE; Alarm12 := FALSE; Alarm13 := FALSE;
	Alarm21 := FALSE; Alarm22 := FALSE; Alarm23 := FALSE;
	Alarm31 := FALSE; Alarm32 := FALSE; Alarm33 := FALSE;
	Alarm40 := FALSE; Alarm41 := FALSE; Alarm42 := FALSE; Alarm43 := FALSE; Alarm44 := FALSE; Alarm45 := FALSE; Alarm46 := FALSE; Alarm47 := FALSE;
	Alarm50 := FALSE; Alarm51 := FALSE; Alarm52 := FALSE; Alarm53 := FALSE; Alarm54 := FALSE; Alarm55 := FALSE; Alarm56 := FALSE; Alarm57 := FALSE;
	Alarm58 := FALSE; Alarm59 := FALSE; Alarm5A := FALSE; Alarm5B := FALSE; Alarm5C := FALSE; Alarm5D := FALSE; Alarm5E := FALSE;
END_IF;

alarmState := INT_TO_BOOL(D0);
attentionState := INT_TO_BOOL(D1) OR INT_TO_BOOL(D2) OR INT_TO_BOOL(D3) OR INT_TO_BOOL(D4) OR INT_TO_BOOL(D5);

lightAlarm := alarmState;
lightAttention := stepStartMotors<>0 OR stepPneumaticPositioning<>0 OR attentionState;

Alarm01 := NOT thermicOk;	(* Сработала тепловая защита *)
Alarm02 := NOT airPressureOk; (* Низкое давление сжатого воздуха *)
Alarm03 := NOT controlVoltageOk; (* Выключено управляющее напряжение *)
Alarm04 := NOT buttonEnable;	 (* Нажата кнопка СТОП *)
Alarm09 := bypassKey; (* Повёрнут ключ отлючения цепочки безопасности *)

(* Одновременно сработали датчики верхнего и нижнего положения шпинделей 1-2-3 *)
SET(spindle1.sensorUp AND spindle1.sensorDown, Alarm11);
SET(spindle2.sensorUp AND spindle2.sensorDown, Alarm21);
SET(spindle3.sensorUp AND spindle3.sensorDown, Alarm31);

(* Ошибка датчиков горизонтального положения шпинделей 1-2-3 *)
TONspindle1Out(IN:= (spindle1.valveIn XOR NOT spindle1.sensorOut) , PT:= T#10s ,Q:= Alarm12 );
TONspindle2Out(IN:= (spindle2.valveIn XOR NOT spindle2.sensorOut) , PT:= T#10s ,Q:= Alarm22 );
TONspindle3Out(IN:= (spindle3.valveIn XOR NOT spindle3.sensorOut) , PT:= T#10s ,Q:= Alarm32 );

(* Ошибка датчиков вертикального положения шпинделей 1-2-3 *)
TONspindle1Vertical(IN:= (spindle1.valveUp AND NOT spindle1.sensorUp) OR (spindle1.valveDown AND NOT spindle1.sensorDown), PT:= T#10s ,Q:= Alarm13 );
TONspindle2Vertical(IN:= (spindle2.valveUp AND NOT spindle2.sensorUp) OR (spindle2.valveDown AND NOT spindle2.sensorDown), PT:= T#10s ,Q:= Alarm23 );
TONspindle3Vertical(IN:= (spindle3.valveUp AND NOT spindle3.sensorUp) OR (spindle3.valveDown AND NOT spindle3.sensorDown), PT:= T#10s ,Q:= Alarm33 );

(* Ошибка датчиков каретки - Одновременно сработали несколько датчиков *)
SET((BOOL_TO_INT(carriageSensor1)+BOOL_TO_INT(carriageSensor2)+BOOL_TO_INT(carriageSensor3)+BOOL_TO_INT(carriageSensor4)) > 1, Alarm40);
END_PROGRAM

PROGRAM Carriage
VAR
  TONCarriagePressRelease : TON;
  FB_DOUBLE_CLICK_F : FB_DOUBLE_CLICK;
  FB_DOUBLE_CLICK_B : FB_DOUBLE_CLICK;
  TONCarriageF : TON;
  TONCarriageAlarmF : TON;
  TONCarriageAlarmB : TON;
  TONCarriageB : TON;
END_VAR
(* Прижим детали на каретке *)
IF MEP(buttonPress) AND NOT carriageMoving THEN
	pressCarriageValveDown := INV(pressCarriageValveDown);
	pressCarriageValveUp := INV(pressCarriageValveDown);
END_IF;

(* Отпустить прижим во время цикла перегрузки с каретки под роликовый транспортёр *) 
TONCarriagePressRelease(IN:=(stepAuto=60) , PT:=hmiPar3);
IF TONCarriagePressRelease.Q THEN
	pressCarriageValveDown := FALSE;
	pressCarriageValveUp := INV(pressCarriageValveDown);
END_IF;

RST(pressCarriageValveDown, Alarm53); (* Сброс аварии - Попытка запуска цикла обработки с не прижатой деталью *)



(* ========================================================================================================= *)
(* ========================================= Перемещение каретки ========================================== *)

(* Быстрое двойное нажатие в ручном режиме *)
IF manualMode AND spindle0NotMiddle THEN
	FB_DOUBLE_CLICK_F(IN:= buttonCarriageForward , PERIOD:= T#1s);
	SET(FB_DOUBLE_CLICK_F.Q, manCarriageMoveToSensor4); (* Перемещение каретки влево к датчику 1 *)

	FB_DOUBLE_CLICK_B(IN:= buttonCarriageBackward , PERIOD:= T#1s);
	SET(FB_DOUBLE_CLICK_B.Q, manCarriageMoveToSensor1);  (* Перемещение каретки вправо к датчику 4 *)
END_IF;

IF buttonCarriageForward OR buttonCarriageBackward OR NOT manualMode OR NOT buttonEnable OR NOT safetyCircuiteOk THEN
	manCarriageMoveToSensor1 := FALSE;
	manCarriageMoveToSensor4 := FALSE;
END_IF;
RST(carriageSensor4, manCarriageMoveToSensor4);
RST(carriageSensor1, manCarriageMoveToSensor1);
	
(* Условия движения каретки вперёд *)
carriageNeedForward := FALSE;
Alarm49 := FALSE;
IF (manualMode AND (buttonCarriageForward OR manCarriageMoveToSensor4)) OR (automaticMode AND carriageAutoForward) THEN
	carriageNeedForward := NOT carriageSensor4;
	Alarm49 := carriageSensor4;
END_IF;
			
(* Условия движения каретки назад *)
carriageNeedBackward := FALSE;
Alarm48 := FALSE;
IF (manualMode AND (buttonCarriageBackward OR manCarriageMoveToSensor1)) OR (automaticMode AND carriageAutoBackward) THEN
	carriageNeedBackward := NOT carriageSensor1;
	Alarm48 := carriageSensor1;
END_IF;

(* Авария - Ручное управление кареткой в Автоматическом режиме *)
IF NOT manualMode AND (buttonCarriageForward OR buttonCarriageBackward) THEN
	Alarm5B := TRUE;
END_IF;
RST(manualMode, Alarm5B);

carriageMoveEnable := (carriageNeedForward XOR carriageNeedBackward) AND ((NOT Alarm45 AND NOT Alarm46) OR bypassKey);

(* Включение тормозного резитора *)
SET(MEP(carriageSensor4), carriageMotorBrake);
RST(carriageMoveEnable, carriageMotorBrake);

(* Включение мотора каретки *)
carriageMotorForward := FALSE;
carriageMotorBackward := FALSE;

TONCarriageF.IN:=FALSE;
TONCarriageB.IN:=FALSE;
IF carriageMoveEnable AND NOT carriageMotorBrake THEN
	IF NOT carriageMotorBackward THEN TONCarriageF(IN:=carriageNeedForward); END_IF; (* Задержка включения мотора вперёд *)
	IF NOT carriageMotorForward THEN TONCarriageB(IN:=carriageNeedBackward); END_IF; (* Задержка включения мотора назад *)
END_IF;
carriageMotorForward := TONCarriageF.Q;
carriageMotorBackward := TONCarriageB.Q;
TONCarriageF(PT:= T#1s);
TONCarriageB(PT:= T#1s);

carriageMoving := carriageMoveEnable OR carriageMotorForward OR carriageMotorBackward;

TONCarriageAlarmF(IN:=carriageMotorForward, PT:= hmiPar6);
IF TONCarriageAlarmF.Q THEN
	Alarm45 := TRUE;
	Alarm44 := TRUE;
END_IF;

TONCarriageAlarmB(IN:=carriageMotorBackward, PT:= hmiPar6);
IF TONCarriageAlarmB.Q THEN
	Alarm46 := TRUE;
	Alarm41 := TRUE;
END_IF;



(* Скорость движения каретки *)
CASE carriageSpeed OF
	3: (* Выбор быстрой скорости *)
		carriageSpeedFast := TRUE;
		carriageSpeedSlow := INV(carriageSpeedFast); carriageSpeedWork := INV(carriageSpeedFast);
	5: (* Выбор скорости обработки резой *)
		carriageSpeedWork := TRUE;
		carriageSpeedSlow := INV(carriageSpeedWork); carriageSpeedFast := INV(carriageSpeedWork);
	ELSE (* Выбор медленной скорости *)
		carriageSpeedSlow := TRUE; carriageSpeedFast := INV(carriageSpeedSlow); carriageSpeedWork := INV(carriageSpeedSlow);
END_CASE;


(* Проверка датчиков каретки *)
IF MEP(carriageSensor1) THEN sensorPositionCurrent := 1;
ELSIF MEP(carriageSensor2) THEN sensorPositionCurrent := 2;
ELSIF MEP(carriageSensor3) THEN sensorPositionCurrent := 3;
ELSIF MEP(carriageSensor4) THEN sensorPositionCurrent := 4;
END_IF;

IF (MEP(carriageSensor1) OR MEP(carriageSensor2) OR MEP(carriageSensor3) OR MEP(carriageSensor4)) THEN
	IF sensorPositionPrev=0 THEN sensorPositionPrev := sensorPositionCurrent; (* Выполняется один раз при срабатывании одного из датчиков каретки *)
	ELSIF ABS(sensorPositionPrev - sensorPositionCurrent) > 1 THEN
		IF (sensorPositionPrev=1 AND sensorPositionCurrent=3) OR (sensorPositionPrev=3 AND sensorPositionCurrent=1) THEN
			Alarm42 := TRUE; (* Не сработал датчик 2 *)
		ELSIF (sensorPositionPrev=1 AND sensorPositionCurrent=4) OR (sensorPositionPrev=4 AND sensorPositionCurrent=1) THEN
			Alarm42 := TRUE; Alarm43 := TRUE; (* Не сработали датчики 2 и 3 *)
		ELSIF (sensorPositionPrev=2 AND sensorPositionCurrent=4) OR (sensorPositionPrev=4 AND sensorPositionCurrent=2) THEN
			Alarm43 := TRUE; (* Не сработал датчик 3 *)
		END_IF;
	ELSE sensorPositionPrev := sensorPositionCurrent;
	END_IF;
END_IF;

IF NOT buttonEnable THEN sensorPositionPrev := 0; END_IF;
END_PROGRAM

PROGRAM Automatic_Cycles
VAR
  stepFirstRun : BOOL;
  TONSlowDown : TON;
  fbMeasureSpeed : FB_MEASURE_SPEED;
  TP_1 : TP;
END_VAR
IF NOT buttonEnable OR NOT safetyCircuiteOk OR NOT automaticMode OR Alarm41 OR Alarm42 OR Alarm43 OR Alarm44 THEN
	stepAuto := 0;
	rollersTransporterAuto := FALSE;
END_IF;

IF MEP(buttonStart) OR MEP(buttonStart2) OR MEP(buttonQuickCut) THEN
	SET(NOT automaticMode, Alarm5A); (* Попытка запуска автоматического цикла не в автоматическом режиме *)
	SET(machineBusy AND stepAuto<>0 AND stepAuto<>40, Alarm5C);	(* Попытка запуска автоматического цикла во время выполнения исполнения другого цикла *)
	SET(machineBusy AND MEP(buttonQuickCut), Alarm5C);	(* Попытка запуска автоматического цикла во время выполнения исполнения другого цикла *)
	SET(stepPneumaticPositioning<>0,  Alarm50); (* Попытка запуска автоматического цикла во время расстановки узлов *)
	SET(stepStartMotors<>0 , Alarm51); (* Попытка запуска автоматического цикла во время запуска моторов *)
END_IF;

RST(automaticMode, Alarm5A);

SET((NOT motorsDovetail AND NOT motorsProfile) AND (MEP(buttonStart) OR MEP(buttonStart2)), Alarm52);
RST(motorsDovetail OR motorsProfile, Alarm52);

SET(NOT motorsProfile AND MEP(buttonStart2), Alarm5E);
RST(motorsProfile, Alarm5E);

IF automaticMode AND NOT machineBusy THEN
	IF motorsDovetail AND MEP(buttonStart) THEN stepAuto := 10;
	ELSIF motorsDovetail AND motorsProfile AND MEP(buttonStart2) THEN stepAuto := 10;
	ELSIF NOT motorsDovetail AND motorsProfile AND (MEP(buttonStart) OR MEP(buttonStart2)) THEN stepAuto := 100;
	ELSIF MEP(buttonQuickCut) THEN stepAuto := 300;
	END_IF;
END_IF;


CASE stepAuto OF
	0:
		carriageAutoForward := FALSE;
		carriageAutoBackward := FALSE;
		Alarm5C := FALSE;
		stepFirstRun := TRUE;
		lightCycleRun := FALSE;
		carriageSpeed := 1;
		TONSlowDown(IN:=FALSE);

	10: (* Подготовка к автоматическому циклу обработки торца. Перемещение к датчику 1 *)
		IF (stepFirstRun AND carriageSensor1) THEN
			IF pressCarriageValveDown THEN
				IF buttonStart2 AND motorsProfile THEN stepAuto := 50; ELSE stepAuto := 20; END_IF;		
			ELSE
				Alarm53 := TRUE;
				stepAuto := 0;
			END_IF;
			
		ELSE 
			stepFirstRun := FALSE;
			IF spindle0NotMiddle THEN
				carriageAutoBackward := TRUE; carriageSpeed := 1;
				IF carriageSensor1 THEN stepAuto := 0; END_IF;
			ELSE
			 	Alarm47 := TRUE;
			 	stepAuto := 0;
			 END_IF;
		END_IF;

	20: (* Автоматический цикл обработки торца *)
		carriageAutoForward := TRUE;
		IF hmiPar11 THEN carriageSpeed := 3; ELSE carriageSpeed := 1; END_IF;
		IF MEF(carriageSensor2) THEN stepAuto := 25; END_IF;
		fbMeasureSpeed(pulseIN1:= MEF(carriageSensor1) , pulseIN2:= MEF(carriageSensor2) , MM:= distanceS1S2 , Q := speedCut);
		fbMeasureSpeed(pulseIN1:=MEF(carriageSensor2));
		
	25: (* Замедление в зоне работы фрезы *)
		carriageSpeed := 5;
		IF carriageSensor3 THEN
			carriageAutoForward := FALSE;
			stepAuto := 30;
		END_IF;
		PLF(TRUE, M1);
		fbMeasureSpeed(pulseIN2:= MEP(carriageSensor3) , MM:= distanceS2S3, Q := speedMill);
		
	30: (* Возврат после первой стадии обработки торца *)
		carriageAutoBackward := TRUE; carriageSpeed := 3;
		IF carriageSensor2 THEN stepAuto := 35; END_IF;

	35: (* Замедление каретки после датчика 2 *)
		TONSlowDown.IN := TRUE;
		IF TONSlowDown.Q THEN carriageSpeed := 1; END_IF;
		IF carriageSensor1 THEN
			carriageAutoBackward := FALSE;
			TONSlowDown.IN:= FALSE;
			stepAuto := 0; (* Завершить цикл, если шпиндели 1-2-3 выключены *)
			IF motorsProfile THEN stepAuto := 40; END_IF;
		END_IF;
		TONSlowDown(PT:= hmiPar1);

	40: (* Разворот детали *)
		IF buttonStart OR buttonStart2 THEN
			IF pressCarriageValveDown THEN stepAuto := 50;
			ELSE Alarm53 := TRUE; END_IF;
		END_IF;

	50: (* Вторая стадия обработки торца с разгрузкой под ролики *)
		carriageAutoForward := TRUE;
		IF hmiPar11 THEN carriageSpeed := 3; ELSE carriageSpeed := 1; END_IF;
		IF MEF(carriageSensor2) THEN stepAuto := 55; END_IF;

	55: (* Замедление в зоне работы фрезы *)
		carriageSpeed := 5;
		IF carriageSensor3 THEN stepAuto := 57; END_IF;

	57: (* Медленная скорость перед датчиком 4 *)
		carriageSpeed := 1;
		IF carriageSensor4 THEN
			carriageAutoForward := FALSE;
			stepAuto := 60;
		END_IF;
		
	60: (* Разгрузка детали под ролики *)
		rollersTransporterAuto := TRUE;
		IF MEF(pieceInStart) THEN stepAuto := 70; END_IF;

	70: (* Возврат каретки к датчику 1 *)
		carriageAutoBackward := TRUE; carriageSpeed := 3;
		IF carriageSensor2 THEN stepAuto := 75; END_IF;

	75:  (* Завершение автоматического цикла *)
		TONSlowDown.IN := TRUE;
		IF TONSlowDown.Q THEN carriageSpeed := 1; END_IF;
		IF carriageSensor1 THEN
			stepAuto := 0;
			TONSlowDown.IN := FALSE;
		END_IF;
		TONSlowDown(PT:= hmiPar1);



	100: (* Подготовка к автоматическому циклу только со шпинделями 1-2-3 *)
		IF carriageSensor4 THEN
			carriageAutoForward := FALSE;
			stepAuto := 110;
		ELSE 
			IF spindle0NotMiddle THEN
				carriageAutoForward := TRUE;
				carriageSpeed := 1;
			ELSE
				Alarm47 := TRUE;
				stepAuto := 0;
			END_IF;
		END_IF;

	110: (* Автоматический цикл только со шпинделями 1-2-3 *)
		rollersTransporterAuto := TRUE;



	300: (* Подготовка к быстрой торцовке Quick Cut *)
		IF stepFirstRun AND carriageSensor1 THEN stepAuto := 310;
		ELSE
			stepFirstRun := FALSE;
			IF spindle0NotMiddle THEN
				carriageAutoBackward := TRUE;
				IF carriageSensor1 THEN stepAuto := 0; END_IF;
			END_IF;
		END_IF;

	310: (* Быстрая торцовка Quick Cut *)
		IF pressCarriageValveDown THEN
			carriageAutoForward := TRUE;
			sawCarriageMotor := TRUE;
			IF hmiPar11 THEN carriageSpeed := 3; ELSE carriageSpeed := 1; END_IF;
			IF MEF(carriageSensor2) THEN
				sawCarriageMotor := FALSE;
				carriageAutoForward := FALSE;
				stepAuto := 320;
			END_IF;
		ELSIF NOT pressCarriageValveDown THEN
			Alarm53 := TRUE;
			stepAuto := 0;
		END_IF;
		
		fbMeasureSpeed(pulseIN1:= MEF(carriageSensor1) , pulseIN2:= MEF(carriageSensor2) , MM:= distanceS1S2 , Q := speedCut);

	320: (* Возврат после Quick Cut к датчику 1 *)
		IF hmiPar10 THEN 
			carriageAutoBackward := TRUE;
			carriageSpeed := 3;
		ELSE stepAuto := 0; END_IF;
		IF carriageSensor2 THEN stepAuto := 325; END_IF;

	325: (* Замедление каретки после датчика 2 *)
		TONSlowDown.IN := TRUE;
		IF TONSlowDown.Q THEN carriageSpeed := 1; END_IF;
		IF carriageSensor1 THEN
			stepAuto := 0;
			TONSlowDown.IN := FALSE;
		END_IF;
		TONSlowDown(PT:= hmiPar1);
		
END_CASE;


IF rollersTransporterAuto AND (stepAuto<100) THEN
	TP_1(IN:= MEF(pieceInEnd) ,PT:= hmiPar5 );
	RST(MEF(TP_1.Q), rollersTransporterAuto);
END_IF;

IF stepAuto <> 0 THEN
	lightCycleRun := TRUE;
END_IF;

machineBusy := stepAuto<>0 OR stepPneumaticPositioning<>0 OR stepStartMotors<>0;
END_PROGRAM

FUNCTION_BLOCK FB_MEASURE_SPEED
VAR_INPUT
  pulseIN1 : BOOL;
  pulseIN2 : BOOL;
  MM : INT;
END_VAR
VAR
  timeStart : TIME;
  timeEnd : TIME;
END_VAR
VAR_OUTPUT
  Q : INT;
END_VAR
(* Измерение скорости движения каретки *)
IF pulseIN1 THEN
	timeStart := plcRunTime;
END_IF;

IF pulseIN2 THEN
	timeEnd := plcRunTime;

	IF timeEnd > timeStart THEN
		Q := DINT_TO_INT( INT_TO_DINT(MM)*60*10/TIME_TO_DINT(timeEnd-timeStart));
	END_IF;

END_IF;
END_FUNCTION_BLOCK
